ORGANIZATION_BLOCK "Main"
TITLE = "Main Program Sweep (Cycle)"
{ S7_Optimized_Access := 'TRUE' }
VERSION : 0.1

BEGIN
	"Block_1_DB"();
	"Block_2_FBD_DB"();

END_ORGANIZATION_BLOCK

